FUNCTION_BLOCK FB_PackMLControl_Auto EXTENDS FB_PackMLControl
VAR_INPUT
	ap_fbEvents : POINTER TO ARRAY [0..1023] OF POINTER TO FB_DiscreteEvents;	
END_VAR
VAR_OUTPUT
END_VAR
VAR
	state : E_PackMLStates := E_PackMLStates.idle;
	ap_fbEventsIdle : ARRAY [0..0] OF POINTER TO FB_DiscreteEvents;		
	ap_fbEventsStarting : ARRAY [0..0] OF POINTER TO FB_DiscreteEvents;		
	ap_fbEventsExecute : ARRAY [0..0] OF POINTER TO FB_DiscreteEvents;	
	ap_fbEventsStop : ARRAY [0..254] OF POINTER TO FB_DiscreteEvents;			
END_VAR

METHOD PROTECTED _mapping : HResult
VAR_INPUT
END_VAR
ap_fbEventsIdle[0] := ap_fbEvents^[0];
ap_fbEventsStarting[0] := ap_fbEvents^[1];
ap_fbEventsExecute[0] := ap_fbEvents^[5];
END_METHOD

METHOD PUBLIC M_Aborted : HResult
VAR_INPUT
END_VAR
END_METHOD

METHOD PUBLIC M_Aborting : HResult
VAR_INPUT
END_VAR
END_METHOD

METHOD PUBLIC M_Complete : HResult
VAR_INPUT
	lastResult : HResult;
END_VAR
VAR_OUTPUT
	abort : BOOL;
END_VAR
VAR_INST
	_fbResult : FB_ResultHelper_V2_1;	
	_lastResult : HRESULT;
	_state : POINTER TO DINT;
END_VAR
_state := ADR(state_complete);
IF _fbResult.M_MethodResult(M_Complete,lastResult,ADR(_lastResult)) = FALSE THEN
	RETURN;
END_IF

IF _fbResult.P_MethodResult = E_Result.S_OK THEN
	_state^ := 0;
END_IF

_fbResult.P_MethodResult := MPM_FBResult.E_Result.S_OK;
END_METHOD

METHOD PUBLIC M_Completing : HREsult
VAR_INPUT
	lastResult : HResult;
END_VAR
VAR_OUTPUT
	abort : BOOL;	
	stop : BOOL;
END_VAR
VAR_INST
	_fbResult : FB_ResultHelper_V2_1;	
	_lastResult : HRESULT;
	_state : POINTER TO DINT;
END_VAR
_state := ADR(state_completing);
IF _fbResult.M_MethodResult(M_Completing,lastResult,ADR(_lastResult)) = FALSE THEN
	RETURN;
END_IF

IF _fbResult.P_MethodResult = E_Result.S_OK THEN
	_state^ := 0;
END_IF

_fbResult.P_MethodResult := MPM_FBResult.E_Result.S_OK;
END_METHOD

METHOD PUBLIC M_Execute : HResult
VAR_INPUT
	lastResult : HResult;
END_VAR
VAR_OUTPUT
	stop : BOOL;
	suspend : BOOL;
	hold : BOOL;
END_VAR
VAR_INST
	_fbResult : FB_ResultHelper_V2_1;	
	_lastResult : HRESULT;
	_state : POINTER TO DINT;
	_ap_fbEventsExecute0_Result : HResult;
END_VAR
_state := ADR(state_execute);
IF _fbResult.M_MethodResult(M_Execute,lastResult,ADR(_lastResult)) = FALSE THEN
	RETURN;
END_IF

IF _fbResult.P_MethodResult = E_Result.S_OK THEN
	_state^ := 0;
END_IF

_fbResult.P_MethodResult := ap_fbEventsExecute[0]^.M_Execute(_fbResult.P_MethodResult);
END_METHOD

METHOD PUBLIC M_ExecuteControl : HResult //needs to run all the time
VAR_INPUT
END_VAR
VAR
	loopCounter : DINT;
	currentState : E_PackMLStates;
END_VAR
_mapping();
currentState := state;
FOR loopCounter := 0 TO 20 BY 1 DO 
	CASE state OF
		E_PackMLStates.aborted:
			M_Aborted();
		E_PackMLStates.aborting:
			M_Aborting();
		E_PackMLStates.complete:
			stateMachineResult := M_Complete(stateMachineResult);
			IF stateMachineResult = MPM_FBResult.E_Result.S_OK THEN
				state := E_PackMLStates.complete;
			END_IF		
		E_PackMLStates.completing:	
			stateMachineResult := M_Completing(stateMachineResult);
			IF stateMachineResult = MPM_FBResult.E_Result.S_OK THEN
				state := E_PackMLStates.idle;
			END_IF					
		E_PackMLStates.execute:	
			stateMachineResult := M_Execute(stateMachineResult);	
			IF stateMachineResult = MPM_FBResult.E_Result.S_OK THEN
				state := E_PackMLStates.completing;
			END_IF			
		E_PackMLStates.held:	
			M_Held();	
		E_PackMLStates.holding:	
			M_Holding();		
		E_PackMLStates.idle:	
			stateMachineResult := M_Idle(stateMachineResult);		
			IF stateMachineResult = MPM_FBResult.E_Result.S_WORKING AND start = TRUE THEN
				stateMachineResult := MPM_FBResult.E_Result.S_OK;
				start := FALSE;
				state := E_PackMLStates.starting;
			END_IF	
		E_PackMLStates.starting:	
			stateMachineResult := M_Starting(stateMachineResult);
			IF stateMachineResult = MPM_FBResult.E_Result.S_OK THEN
				state := E_PackMLStates.execute;
			END_IF		
		E_PackMLStates.stopped:	
			M_Stopped();	
		E_PackMLStates.stopping:	
			M_Stopping();
		E_PackMLStates.suspdending:	
			M_Suspending();		
		E_PackMLStates.suspended:	
			M_Suspended();	
		E_PackMLStates.un_holding:	
			M_Un_Holding();			
		E_PackMLStates.un_suspsending:	
			M_Un_Suspending();					
	END_CASE
	
	IF currentState = state THEN // if state didnt change
	 	EXIT;
	ELSE // if state changed
		currentState := state;
	END_IF
	
END_FOR
END_METHOD

METHOD PUBLIC M_Held : HResult
VAR_INPUT
END_VAR
VAR_OUTPUT
	abort : BOOL;
	stop : BOOL;
END_VAR
END_METHOD

METHOD PUBLIC M_Holding : HResult
VAR_INPUT
END_VAR
VAR_OUTPUT
	abort : BOOL;
	stop : BOOL;
END_VAR
END_METHOD

METHOD PUBLIC M_Idle : HResult
VAR_INPUT
	lastResult : HResult;
END_VAR
VAR_OUTPUT
	abort : BOOL;
END_VAR
VAR_INST
	_fbResult : FB_ResultHelper_V2_1;	
	_lastResult : HRESULT;
	_state : POINTER TO DINT;
END_VAR
_state := ADR(state_idle);
IF _fbResult.M_MethodResult(M_Idle,lastResult,ADR(_lastResult)) = FALSE THEN
	RETURN;
END_IF

_fbResult.P_MethodResult := ap_fbEventsIdle[0]^.M_Execute(_fbResult.P_MethodResult);
END_METHOD

METHOD PUBLIC M_Resetting : HResult
VAR_INPUT
END_VAR
VAR_OUTPUT
	abort : BOOL;
	stop : BOOL;
END_VAR
END_METHOD

METHOD M_Starting : HResult
VAR_INPUT
	lastResult : HResult;
END_VAR
VAR_OUTPUT
	abort : BOOL;
END_VAR
VAR_INST
	_fbResult : FB_ResultHelper_V2_1;	
	_lastResult : HRESULT;
	_state : POINTER TO DINT;
END_VAR
_state := ADR(state_starting);
IF _fbResult.M_MethodResult(M_Starting,lastResult,ADR(_lastResult)) = FALSE THEN
	RETURN;
END_IF

IF _fbResult.P_MethodResult = E_Result.S_OK THEN
	_state^ := 0;
END_IF

_fbResult.P_MethodResult := ap_fbEventsStarting[0]^.M_Execute(_fbResult.P_MethodResult);
END_METHOD

METHOD PUBLIC M_Stopped : HResult
VAR_INPUT
	
END_VAR
VAR_OUTPUT
	abort : BOOL;
END_VAR
END_METHOD

METHOD PUBLIC M_Stopping : HResult
VAR_INPUT
END_VAR
VAR_OUTPUT
	abort : BOOL;
END_VAR
END_METHOD

METHOD PUBLIC M_Suspended : HREsult
VAR_INPUT
END_VAR
VAR_OUTPUT
	abort : BOOL;
	stop : BOOL;
END_VAR
END_METHOD

METHOD PUBLIC M_Suspending : HREsult
VAR_INPUT
END_VAR
VAR_OUTPUT
	abort : BOOL;
	stop : BOOL;
END_VAR
END_METHOD

METHOD PUBLIC M_Un_Holding : HREsult
VAR_INPUT
END_VAR
VAR_OUTPUT
	abort : BOOL;
	stop : BOOL;
END_VAR
END_METHOD

METHOD PUBLIC M_Un_Suspending : HREsult
VAR_INPUT
END_VAR
VAR_OUTPUT
	abort : BOOL;
	stop : BOOL;
END_VAR
END_METHOD

END_FUNCTION_BLOCK

(* stored: Version 1.1.0.1, ProductVersion 3.1.4024.12
   POU FB_PackMLControl_Auto: Id {c5833f27-92ed-4a89-a91d-67d8b5f3dd79}, SpecialFunc None
   Method _mapping: Id {95fbdf69-4d70-4cf0-a04e-f41a3e57e609}
   Method M_Aborted: Id {78c335fe-acda-4014-bd30-8b866a0d5e43}
   Method M_Aborting: Id {3444003e-e921-4628-8bfe-b7455b07afae}
   Method M_Complete: Id {e5efc557-b039-48cd-8059-7b3d06b26dd5}
   Method M_Completing: Id {c33a5f9d-3834-4555-89e4-e4cada89ab06}
   Method M_Execute: Id {4ec5b464-8a5b-449b-bc5c-de54e9781e20}
   Method M_ExecuteControl: Id {4df9f829-aaf0-41eb-9d68-385cbd1434e7}
   Method M_Held: Id {5f4f9a6e-7b10-4172-b2ba-372008d57881}
   Method M_Holding: Id {9b8e953a-67a9-4124-a710-543f9bcd787e}
   Method M_Idle: Id {a2ad968b-e06b-4127-b93d-485aac283c9f}
   Method M_Resetting: Id {1d9ec857-5dd6-4bb9-b218-cc4502e6f587}
   Method M_Starting: Id {0a584554-f30b-440d-bb06-5ff45cfb6c10}
   Method M_Stopped: Id {6f1dabcb-5a75-484d-bf5e-d7f7a44ed766}
   Method M_Stopping: Id {a2477e6e-33d5-4e37-bed5-b0a371e17491}
   Method M_Suspended: Id {18c1fede-7d2b-47e6-95f4-b091adaa6a30}
   Method M_Suspending: Id {9c59d699-c5c5-475b-aa59-8610ed99caaa}
   Method M_Un_Holding: Id {2ef0d78f-60a7-40e0-9514-17a12d1dbc9e}
   Method M_Un_Suspending: Id {2712b190-017e-4147-be22-b22e015dc8b8} *)
